{attribute 'GeneratedUsingTerminal: IODEVICETYPE_ETHERCATPROT'}
{attribute addProperty BoxType "IODEVICETYPE_ETHERCATPROT"}
{attribute addProperty Id "Term_9_EK1100Term_9_EK1100_00369A35110Term_14_EK1100Term_14_EK1100_023262FB285SyncUnitsSyncUnits_1397309536InputsInputs_A65FACA410OutputsOutputs_23C0ED1D6InfoDataInfoData_E68C61CD28"}
{attribute addProperty CRC "2705793974"}
{attribute addProperty Size "475"}
TYPE Device_4_EtherCAT_A14723B6 :
STRUCT
	{attribute addProperty Name "Term_9_EK1100"}
	{attribute addProperty PreviousPort "Device 4 (EtherCAT) : Master"}
	Term_9_EK1100 : Term_9_EK1100_00369A35;
	{attribute addProperty Name "Term_14_EK1100"}
	{attribute addProperty PreviousPort "Term 13 (EK1110) : B"}
	Term_14_EK1100 : Term_14_EK1100_023262FB;
	{attribute addProperty Name "SyncUnits"}
	SyncUnits : SyncUnits_13973095;
	{attribute addProperty Name "Inputs"}
	Inputs : TcoIo.Inputs_A65FACA4;
	{attribute addProperty Name "Outputs"}
	Outputs : TcoIo.Outputs_23C0ED1D;
	{attribute addProperty Name "InfoData"}
	InfoData : TcoIo.InfoData_E68C61CD;
END_STRUCT
END_TYPE

(* stored: Version 1.2.0.0, ProductVersion 3.1.4024.9
   DUT Device_4_EtherCAT_A14723B6: Id {14258f1a-330b-0401-2e9b-ca2d1f8ac47c} *)
